TYPE ST_EventsAssigment :
STRUCT
	
	sEventText							: STRING(255);
	sSolution							: STRING(255);
END_STRUCT
END_TYPE

(* stored: Version 1.1.0.1, ProductVersion 3.1.4024.13
   DUT ST_EventsAssigment: Id {86b7b955-b4d5-45eb-a3be-b18d5212c670} *)
